// TIA Portal V16 export
// export: Created 2023-09-25T11:31:55.5549636Z, ExportSetting WithDefaults, DisplayName Totally Integrated Automation Portal, DisplayVersion V16 Update 6, DisplayName TIA Portal Version Control Interface, DisplayVersion V16 Update 2, DisplayName TIA Portal Openness, DisplayVersion V16 Update 6, DisplayName STEP 7 Professional, DisplayVersion V16 Update 6, DisplayName STEP 7 Safety, DisplayVersion V16, DisplayName WinCC Advanced, DisplayVersion V16 Update 6
DATA_BLOCK "dbTable of value Hz"   // DB59
TITLE = Table of value Hz manual instruction
{ S7_Optimized_Access := 'TRUE' }
AUTHOR : rtecmer
VERSION : 0.1
// tabela z wartościami Hz przekazywanymi w instrukcji manualnego sterowania regulatorem PID podczas doączenia kompresora dodatkowego po ustawieniu Set 50Hz
// stored: AutoNumber true, DBAccessibleFromOPCUA true, IsOnlyStoredInLoadMemory false, IsRetainMemResEnabled false, IsWriteProtectedInAS false, MemoryReserve 500
   VAR
      Static_1 : Array[0..20] of Real;
      Static_2 : Array[0..10] of Int;
   END_VAR
BEGIN
   Static_1[0] := 2.0;
   Static_1[1] := 3.0;
   Static_1[2] := 4.0;
   Static_1[3] := 5.0;
   Static_1[4] := 6.0;
   Static_1[5] := 7.0;
   Static_1[6] := 8.0;
   Static_1[7] := 10.0;
   Static_1[8] := 12.0;
   Static_1[9] := 13.0;
   Static_1[10] := 14.0;
   Static_1[11] := 15.0;
   Static_1[12] := 20.0;
   Static_1[13] := 30.0;
   Static_1[14] := 40.0;
   Static_1[15] := 50.0;
   Static_1[16] := 60.0;
   Static_1[17] := 70.0;
   Static_1[18] := 80.0;
   Static_1[19] := 90.0;
   Static_1[20] := 100.0;
   Static_2[0] := 8500;
   Static_2[1] := 9500;
   Static_2[2] := 10000;
   Static_2[3] := 10500;
   Static_2[4] := 11000;
   Static_2[5] := 12000;
   Static_2[6] := 13000;
   Static_2[7] := 19000;
   Static_2[8] := 20500;
   Static_2[9] := 25600;
   Static_2[10] := 27648;
END_DATA_BLOCK
